{attribute 'GeneratedUsingTerminal: ELX4181-0000-0016'}
{attribute addProperty BoxType "ELX4181-0000-0016"}
{attribute addProperty Description "ELX4181 1-channel analog output terminal 0/4...20 mA, single-ended, HART, 16 bit, Ex i"}
{attribute addProperty Physics "KK"}
{attribute addProperty Id "Ch_1Ch_1_29D412892WcStateAT %I*WcState_0B2B16F91InfoDataAT %I*InfoData_90184F0C16"}
{attribute addProperty CRC "155821760"}
{attribute addProperty Size "19"}
TYPE ELX4181_0949A6C0 EXTENDS EtcSlaveTerminalBase_947E5A46 :
STRUCT
	{attribute addProperty Name "Ch_1"}
	Ch_1 : Ch_1_29D41289;
	{attribute addProperty Name "WcState"}
	WcState : WcState_0B2B16F9;
	{attribute addProperty Name "InfoData"}
	InfoData : InfoData_90184F0C;
END_STRUCT
END_TYPE

(* stored: Version 1.2.0.0, ProductVersion 3.1.4024.11
   DUT ELX4181_0949A6C0: Id {2b22bbe1-ed46-444b-a858-0cfe2613a773} *)
